PROGRAM MAIN
VAR
END_VAR

END_PROGRAM

(* stored: Version 1.1.0.1
   POU MAIN: Id {d0c1e160-5bff-4df7-91d5-31a6e1df873d} *)
